{attribute 'GeneratedUsingTerminal: EL7211-0000-0020'}
{attribute addProperty BoxType "EL7211-0000-0020"}
{attribute addProperty Id "FB_PositionAT %I*FB_Position_3FA094ED4DRV_StatuswordAT %I*DRV_Statusword_9B36FDFC2DRV_ControlwordAT %Q*DRV_Controlword_F3F147212DRV_Target_velocityAT %Q*DRV_Target_velocity_08A9583B4WcStateAT %I*WcState_9091E0EB2InfoDataAT %I*InfoData_DEBFC8B711"}
{attribute addProperty CRC "2447262704"}
{attribute addProperty Size "25"}
TYPE EL7211_91DE43F0 EXTENDS EtcSlaveTerminalBase_947E5A46 :
STRUCT
	{attribute addProperty Name "FB_Position"}
	FB_Position : FB_Position_3FA094ED;
	{attribute addProperty Name "DRV_Statusword"}
	DRV_Statusword : DRV_Statusword_9B36FDFC;
	{attribute addProperty Name "DRV_Controlword"}
	DRV_Controlword : DRV_Controlword_F3F14721;
	{attribute addProperty Name "DRV_Target_velocity"}
	DRV_Target_velocity : DRV_Target_velocity_08A9583B;
	{attribute addProperty Name "WcState"}
	WcState : WcState_9091E0EB;
	{attribute addProperty Name "InfoData"}
	InfoData : InfoData_DEBFC8B7;
END_STRUCT
END_TYPE

(* stored: Version 1.2.0.0, ProductVersion 3.1.4024.9
   DUT EL7211_91DE43F0: Id {2e057568-9493-41b1-b46b-3fa5ef825754} *)
